// TIA Portal V19 export
TYPE "C904_VAR_IF_VPI_TYPIC"
   STRUCT
      WRE { ExternalAccessible := 'False'; ExternalVisible := 'False'; ExternalWritable := 'False'} : USInt;   // Actueel actief regime
      BMO_HAND { ExternalAccessible := 'False'; ExternalVisible := 'False'; ExternalWritable := 'False'} : Bool;   // TRUE = Regime handmatig ingesteld via lokale bediening
   END_STRUCT;
END_TYPE
